FUNCTION_BLOCK RunLabelHandler EXTENDS RunUnitSlave
VAR_INPUT
END_VAR
VAR_OUTPUT
END_VAR
VAR
	//File handler
	fbOpen : FB_FileOpen;
	fbWrite : FB_FileWrite;
	fbClose : FB_FileClose;
	fileHandle : UINT;
	filePath : STRING := '';
	fileContent : STRING := '100,2';
	fileBytes : ARRAY[0..15] OF BYTE;
	// communicate with external device
	ioPrinter : POINTER TO  ioBundlePrinterApplicator;
	// Vaccuum
	ioVacuum : POINTER TO ioBundleLabelGripper;
	bVacuumSensor : POINTER TO RunSignal;
	//
	axis : POINTER TO RunAxis;
	//
	gripperVertical : POINTER TO RunCylinder;
	gripperRotate : POINTER TO RunCylinder;
	gripperPressorVertical : POINTER TO RunCylinder;
	gripperPressorPress : POINTER TO RunCylinder;
	shifter : POINTER TO RunCylinder;
	//
	ptCommandReady : POINTER TO ParameterSet;
	ptCommandLabelTake : POINTER TO ParameterSet;
	ptCommandLabelPlace : POINTER TO ParameterSet;
	//
	pressCounter : INT := 0;
	//
	bFirstCycle : bool := false;
END_VAR
VAR PERSISTENT
	bVacuumTimeout : TON;
	pressGoal : INT := 3;
END_VAR

SUPER^();

//into initial state
IF NOT bFirstCycle AND outputState=0 THEN
	NextState := 16#300;
	bFirstCycle := TRUE;
END_IF

CASE outputState OF 
	//-------------------Initializing
	eSpecialStates.INITIAL_BEGIN:
		//all cylinder off
		transitionByte.0 := gripperVertical^.Execute(eCylinderCommands.COMMAND_A);
		transitionByte.1 := gripperRotate^.Execute(eCylinderCommands.COMMAND_A);
		transitionByte.2 := gripperPressorVertical^.Execute(eCylinderCommands.COMMAND_A);
		transitionByte.3 := gripperPressorPress^.Execute(eCylinderCommands.COMMAND_A);
		transitionByte.4 := shifter^.Execute(eCylinderCommands.COMMAND_A);
		bSerialTransition := (transitionByte = 16#1F);
	eSpecialStates.INITIAL_STATE_1:
		IF axis^.ExecuteParameter(ptCommandReady) THEN
			bFirstCycle := FALSE;
			NextState := eSpecialStates.INITIAL_END;
		END_IF
	//-------------------Working
	16#300:
		fbOpen.bExecute:=TRUE;
		bSerialTransition := TRUE;
	16#301:
		bSerialTransition := NOT fbOpen.bBusy;
	16#302:
		fbWrite.bExecute := TRUE;
		bSerialTransition := TRUE;
	16#303:
		bSerialTransition := NOT fbWrite.bBusy;
	16#304:
		fbClose.bExecute := TRUE;
		bSerialTransition := TRUE;
	16#305:
		IF NOT fbClose.bBusy THEN
			NextState:=16#400;
		END_IF
	//-----------------------------
	16#400:
		bSerialTransition := ioPrinter^.prtData;
		IF bSerialTransition THEN
			ioPrinter^.prtStart := TRUE;
		END_IF
	16#401:
		//waiting printer
		bSerialTransition := NOT ioPrinter^.prtEnd AND NOT ioPrinter^.prtData;
		IF bSerialTransition THEN
			ioPrinter^.prtStart := false;
		END_IF
	16#402:
		bSerialTransition := axis^.ExecuteParameter(ptCommandLabelTake);
	16#403:
		bSerialTransition := gripperVertical^.Execute(eCylinderCommands.COMMAND_B);	//down
		IF bSerialTransition THEN
			//generate vacuum
			ioVacuum^.vacuumGripper := TRUE; //on
			ioVacuum^.breakGripper := FALSE;
			//
			bVacuumTimeout.IN :=TRUE;
		END_IF
	16#404:
		bSerialTransition := bVacuumSensor^.debouncedOn;
		IF bSerialTransition THEN
			bVacuumTimeout.IN :=FALSE; //reset
		ELSIF bVacuumTimeout.Q THEN
			//TODO , timeout alarm
		END_IF
	16#405:
		bSerialTransition := gripperVertical^.Execute(eCylinderCommands.COMMAND_A); //up
	16#406:
		IF axis^.ExecuteParameter(ptCommandLabelPlace) THEN
			//up
			NextState := 0; //wait trigger
		END_IF
	//-----------------Tag
	eSpecialStates.SLAVE_ENTER_PROCEDURE:
		bSerialTransition := gripperVertical^.Execute(eCylinderCommands.COMMAND_B); //down
		IF bSerialTransition THEN
			//break vacuum
			ioVacuum^.vacuumGripper := FALSE; //off
			ioVacuum^.breakGripper := TRUE;
		END_IF
	16#201:
		transitionByte.0 := gripperVertical^.Execute(eCylinderCommands.COMMAND_A); //up
		transitionByte.1 := gripperRotate^.Execute(eCylinderCommands.COMMAND_A); //back
		bSerialTransition := (transitionByte = 16#3);
	//----------------Press
	16#202:
		bSerialTransition := shifter^.Execute(eCylinderCommands.COMMAND_B); //tool change
	16#203:
		bSerialTransition := gripperPressorVertical^.Execute(eCylinderCommands.COMMAND_B); //down
	16#204:
		bSerialTransition := gripperPressorPress^.Execute(eCylinderCommands.COMMAND_B);
	16#205:
		IF gripperPressorPress^.Execute(eCylinderCommands.COMMAND_A) THEN
			pressCounter := pressCounter+1;
			
			IF pressCounter >= pressGoal THEN
				//press back-forth
				NextState := 16#230;
			ELSE
				NextState := 16#205;
			END_IF
		END_IF
	//------------Return
	16#230:
		bSerialTransition := gripperPressorVertical^.Execute(eCylinderCommands.COMMAND_A); //up
	16#231:
		bSerialTransition := shifter^.Execute(eCylinderCommands.COMMAND_A); //up
		IF bSerialTransition THEN
			workingSignal^ := FALSE; //off
		END_IF
	16#232:
		//ready
		IF axis^.ExecuteParameter(ptCommandLabelTake) THEN
			pressCounter:=0;
			NextState := 16#400;
		END_IF
END_CASE
bVacuumTimeout(IN:= , PT:= , Q=> , ET=> );


//file 
fbOpen(
	sNetId:= , 
	sPathName:= filePath, 
	nMode:= FOPEN_MODEWRITE, 
	ePath:= , 
	bExecute:= , 
	tTimeout:= , 
	bBusy=> , 
	bError=> , 
	nErrId=> , 
	hFile=> fileHandle);
fbWrite(
	sNetId:= , 
	hFile:= fileHandle, 
	pWriteBuff:= ADR(fileBytes), 
	cbWriteLen:= SIZEOF(fileBytes), 
	bExecute:= , 
	tTimeout:= , 
	bBusy=> , 
	bError=> , 
	nErrId=> , 
	cbWrite=> );
fbClose(
	sNetId:= , 
	hFile:= fileHandle, 
	bExecute:= , 
	tTimeout:= , 
	bBusy=> , 
	bError=> , 
	nErrId=> );

METHOD FB_init : BOOL
VAR_INPUT
	bInitRetains : BOOL; // if TRUE, the retain variables are initialized (warm start / cold start)
	bInCopyCode : BOOL;  // if TRUE, the instance afterwards gets moved into the copy code (online change)
	
	argParent : POINTER TO RunUnitGeneric;
	argSlotBase : POINTER TO MaterialBlock;
	argSlotLast : POINTER TO MaterialBlock;
	
	argWorkingSignal : POINTER TO BOOL;
	
	//devices
	argVacuumSensor : POINTER TO RunSignal;
	
	argAxis : POINTER TO RunAxis;
	//
	argGripperVertical : POINTER TO RunCylinder;
	argGripperRotate : POINTER TO RunCylinder;
	argGripperPressorVertical : POINTER TO RunCylinder;
	argGripperPressorPress : POINTER TO RunCylinder;
	argShifter : POINTER TO RunCylinder;
	//
	argIoPrinter : POINTER TO ioBundlePrinterApplicator;
	argIoVacuum : POINTER TO ioBundleLabelGripper;
END_VAR
VAR CONSTANT
	indexReady : INT := 1;
	indexTake :INT :=2;
	indexPlace : INT :=3;
END_VAR
//initialize 
Parent := argParent;
SlotBase := argSlotBase;
SlotLast := argSlotLast;
//
IF bInitRetains THEN
	NextState := eSpecialStates.INITIAL_BEGIN;
END_IF

workingSignal := argWorkingSignal; //link

//device link
//
axis := argAxis;
//
gripperVertical := argGripperVertical;
gripperRotate := argGripperRotate;
gripperPressorVertical := argGripperPressorVertical;
gripperPressorPress := argGripperPressorPress;
shifter := argShifter;

ptCommandReady := ADR(axis^.ptpCommands[indexReady]);
ptCommandLabelTake := ADR(axis^.ptpCommands[indexTake]);
ptCommandLabelPlace := ADR(axis^.ptpCommands[indexPlace]);

bVacuumSensor := argVacuumSensor;

ioPrinter := argIoPrinter;
ioVacuum := argIoVacuum;
END_METHOD

END_FUNCTION_BLOCK

(* stored: Version 1.1.0.1, ProductVersion 3.1.4022.10
   POU RunLabelHandler: Id {e13915db-12ab-405f-bb1f-0c49fc3dffb2}, SpecialFunc None
   Method FB_init: Id {8e22ea07-e6ac-4cce-a3dd-c0421a83bdd3} *)
